// TwinCAT 3 PLC project Main
// ProgramVersion: 3.1.4023.0
// libraries:
//   Tc2_Standard, * (Beckhoff Automation GmbH)
//   Tc2_System, * (Beckhoff Automation GmbH)
//   Tc3_Module, * (Beckhoff Automation GmbH)
// project tree:
//   / PlcTask.TcTTO
//   POUs/ FB_Conveyor_SFC.TcPOU, FB_Conveyor_ST.TcPOU, FB_Coordinador_SFC.TcPOU, FB_Coordinador_ST.TcPOU, FB_Discharger_SFC.TcPOU, FB_Discharger_ST.TcPOU, FB_Elevator_SFC.TcPOU, FB_Elevator_ST.TcPOU, FB_Object_Template_ST.TcPOU, FB_Object_Template_SFC.TcPOU, MAIN.TcPOU
// real-time tasks:
//   TASK PlcTask: cycle T#10ms, priority 20, ADS port 350

CONFIGURATION Main
    RESOURCE PLC ON TwinCAT3
        TASK PlcTask(INTERVAL := T#10ms, PRIORITY := 20);
        PROGRAM MAIN WITH PlcTask : MAIN;
    END_RESOURCE
END_CONFIGURATION

// ---- POUs/MAIN.TcPOU
PROGRAM MAIN
VAR
	
Coordinador : FB_Coordinador_ST;

END_VAR

Coordinador();

END_PROGRAM

// ---- POUs/FB_Coordinador_ST.TcPOU
FUNCTION_BLOCK FB_Coordinador_ST EXTENDS FB_Object_Template_ST
VAR_INPUT
	//Discharger
	Tray_1 : BOOL; 
	Tray_2 : BOOL;
	
END_VAR
VAR_OUTPUT
	Fail : BOOL;
	B1   : BOOL;
	
END_VAR
VAR
	
	Discharger : FB_Discharger_ST;
	Elevators  : FB_Elevator_ST;
	Conveyors  : FB_Conveyor_ST;
	Production: FB_Coordinador_SFC;
	
END_VAR

IC := Discharger.IC AND Elevators.IC AND Conveyors.IC;
B1 := Selector(Tray_1,Tray_2);

Discharger(Execute:=Production.Discharger_Execute,
			Ack:=Production.Discharger_Ack,
			Reset:=Reset,
			Pause:=Pause,
			Tray_1:=Tray_1,
			Tray_2:=Tray_2
			);
			
Elevators.Elevator_B1 (Execute:=Production.Elevator_B1_Execute,
					  Ack:=Production.Elevator_B1_Ack,
					  SFCReset:=Reset,
					  SFCPause:=Pause,
					  );
					
Elevators.Elevator_B2 (Execute:=Production.Elevator_B2_Execute,
					  Ack:=Production.Elevator_B2_Ack,
					  SFCReset:=Reset,
					  SFCPause:=Pause,
					  );
					  
Elevators.Elevator_S (Execute:=Production.Elevator_S_Execute,
					  Ack:=Production.Elevator_S_Ack,
					  SFCReset:=Reset,
					  SFCPause:=Pause,
					  );
					  
Conveyors.Conveyors_B1  (Execute := Production.Conveyor_B1_Execute,
						Ack := Production.Conveyor_B1_Ack,
						SFCReset := Reset,
						SFCPause := Pause,
						);
						
Conveyors.Conveyors_B2  (Execute := Production.Conveyor_B2_Execute,
						Ack := Production.Conveyor_B2_Ack,
						SFCReset := Reset,
						SFCPause := Pause,
						);

Conveyors.Conveyor_S  (Execute := Production.Conveyor_S_Execute,
						Ack := Production.Conveyor_S_Ack,
						SFCReset := Reset,
						SFCPause := Pause,
						);

METHOD Selector : BOOL
VAR_INPUT
	
	Tray_1 : BOOL;
	Tray_2 : BOOL;

END_VAR
IF Tray_1 THEN
	Selector := TRUE;
ELSIF Tray_2 THEN
	Selector := FALSE;
END_IF
END_METHOD

END_FUNCTION_BLOCK

// ---- POUs/FB_Object_Template_ST.TcPOU
FUNCTION_BLOCK FB_Object_Template_ST
VAR_INPUT
	// Control variables
	Execute: BOOL;
	Ack: BOOL;
	Reset: BOOL; 
	Pause: BOOL;
	// Physical variables
	
END_VAR
VAR_OUTPUT
	//Control variables
	Ready: BOOL;
	Done: BOOL;
	//Physical Variables
	
END_VAR
VAR
	// Initial conditions
	IC: BOOL := TRUE;
END_VAR

END_FUNCTION_BLOCK

// ---- POUs/FB_Discharger_ST.TcPOU
FUNCTION_BLOCK FB_Discharger_ST EXTENDS FB_Object_Template_ST
VAR_INPUT
	Tray_1: BOOL; 
	Tray_2: BOOL;
	dcha_1 AT %I*: BOOL;
	dcha_2 AT %I*: BOOL;
	izda_1 AT %I*: BOOL;
	izda_2 AT %I*: BOOL;
	arriba AT %I*: BOOL;
	abajo  AT %I*: BOOL;
	cogido AT %I*: BOOL;
END_VAR
VAR_OUTPUT
	avanza_1 AT %Q*: BOOL;
	avanza_2 AT %Q*: BOOL;
	baja	 AT %Q*: BOOL;
	coge 	 AT %Q*: BOOL;
	Fail : BOOL;
	Timer : TON;
END_VAR
VAR
	Discharger : FB_Discharger_SFC;
END_VAR

//Define initial conditions
IC := izda_1 AND izda_2 AND arriba AND NOT cogido;
//Declare module
Discharger(Execute:=Execute,
		   Ack:=Ack,
		   SFCReset:=Reset,
		   SFCPause:=Pause,
		   IC:=IC,
		   Tray_1:=Tray_1,
		   Tray_2:=Tray_2,
		   dcha_1:=dcha_1,
		   dcha_2:=dcha_2,
		   izda_1:=izda_1,
		   izda_2:=izda_2,
		   arriba:=arriba,
		   abajo:=abajo,
		   cogido:=cogido,
);
		   
//Declare module actuators
Ready := Discharger.Ready;
Done := Discharger.Done;
avanza_1 := Discharger.avanza_1;
avanza_2 := Discharger.avanza_2;
baja := Discharger.baja;
coge := Discharger.coge;

END_FUNCTION_BLOCK

// ---- POUs/FB_Discharger_SFC.TcPOU
FUNCTION_BLOCK FB_Discharger_SFC EXTENDS FB_Object_Template_SFC
VAR_INPUT
	Tray_1: BOOL;
	Tray_2: BOOL;
	dcha_1: BOOL;
	dcha_2: BOOL;
	izda_1: BOOL;
	izda_2: BOOL;
	arriba: BOOL;
	abajo: BOOL;
	cogido: BOOL;
	Restore: BOOL;
END_VAR
VAR_OUTPUT
	avanza_1: BOOL;
	avanza_2: BOOL;
	baja: BOOL;
	coge: BOOL;
END_VAR
VAR
END_VAR

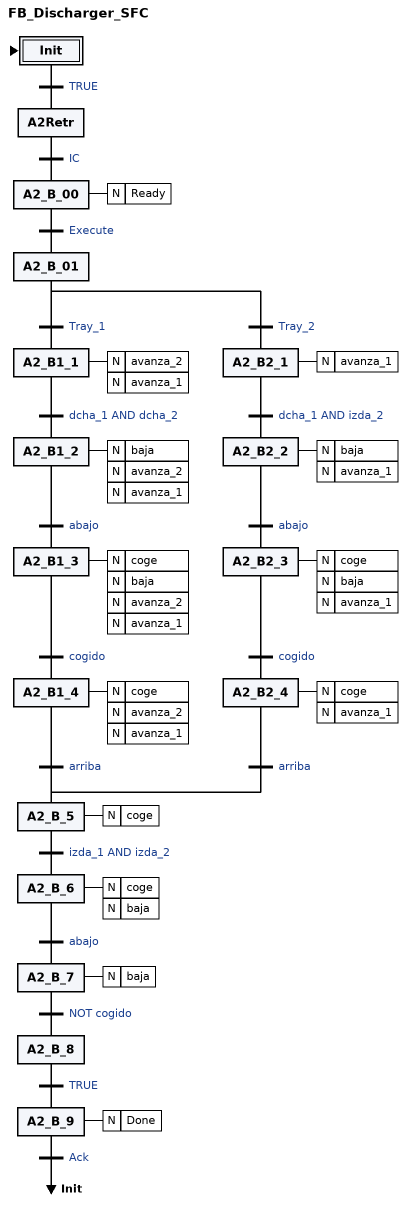
INITIAL_STEP Init:
END_STEP
TRANSITION FROM Init TO A2Retr
    := TRUE;
END_TRANSITION
STEP A2Retr:
END_STEP
TRANSITION FROM A2Retr TO A2_B_00
    := IC;
END_TRANSITION
STEP A2_B_00:
    Ready(N);
END_STEP
TRANSITION FROM A2_B_00 TO A2_B_01
    := Execute;
END_TRANSITION
STEP A2_B_01:
END_STEP
TRANSITION FROM A2_B_01 TO A2_B1_1
    := Tray_1;
END_TRANSITION
STEP A2_B1_1:
    avanza_2(N);
    avanza_1(N);
END_STEP
TRANSITION FROM A2_B1_1 TO A2_B1_2
    := dcha_1 AND dcha_2;
END_TRANSITION
STEP A2_B1_2:
    baja(N);
    avanza_2(N);
    avanza_1(N);
END_STEP
TRANSITION FROM A2_B1_2 TO A2_B1_3
    := abajo;
END_TRANSITION
STEP A2_B1_3:
    coge(N);
    baja(N);
    avanza_2(N);
    avanza_1(N);
END_STEP
TRANSITION FROM A2_B1_3 TO A2_B1_4
    := cogido;
END_TRANSITION
STEP A2_B1_4:
    coge(N);
    avanza_2(N);
    avanza_1(N);
END_STEP
TRANSITION FROM A2_B1_4 TO A2_B_5
    := arriba;
END_TRANSITION
TRANSITION FROM A2_B_01 TO A2_B2_1
    := Tray_2;
END_TRANSITION
STEP A2_B2_1:
    avanza_1(N);
END_STEP
TRANSITION FROM A2_B2_1 TO A2_B2_2
    := dcha_1 AND izda_2;
END_TRANSITION
STEP A2_B2_2:
    baja(N);
    avanza_1(N);
END_STEP
TRANSITION FROM A2_B2_2 TO A2_B2_3
    := abajo;
END_TRANSITION
STEP A2_B2_3:
    coge(N);
    baja(N);
    avanza_1(N);
END_STEP
TRANSITION FROM A2_B2_3 TO A2_B2_4
    := cogido;
END_TRANSITION
STEP A2_B2_4:
    coge(N);
    avanza_1(N);
END_STEP
TRANSITION FROM A2_B2_4 TO A2_B_5
    := arriba;
END_TRANSITION
STEP A2_B_5:
    coge(N);
END_STEP
TRANSITION FROM A2_B_5 TO A2_B_6
    := izda_1 AND izda_2;
END_TRANSITION
STEP A2_B_6:
    coge(N);
    baja(N);
END_STEP
TRANSITION FROM A2_B_6 TO A2_B_7
    := abajo;
END_TRANSITION
STEP A2_B_7:
    baja(N);
END_STEP
TRANSITION FROM A2_B_7 TO A2_B_8
    := NOT cogido;
END_TRANSITION
STEP A2_B_8:
END_STEP
TRANSITION FROM A2_B_8 TO A2_B_9
    := TRUE;
END_TRANSITION
STEP A2_B_9:
    Done(N);
END_STEP
TRANSITION FROM A2_B_9 TO Init
    := Ack;
END_TRANSITION

END_FUNCTION_BLOCK

// ---- POUs/FB_Object_Template_SFC.TcPOU
FUNCTION_BLOCK FB_Object_Template_SFC
VAR_INPUT
	// Control variables
	Execute: BOOL;
	Ack: BOOL;
	SFCReset: BOOL; 
	SFCPause: BOOL;
	IC: BOOL;
	// Physical variables
END_VAR
VAR_OUTPUT
	//Control variables
	Ready: BOOL;
	Done: BOOL;
	//Physical Variables
END_VAR
VAR
END_VAR

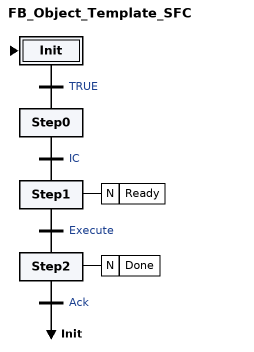
INITIAL_STEP Init:
END_STEP
TRANSITION FROM Init TO Step0
    := TRUE;
END_TRANSITION
STEP Step0:
END_STEP
TRANSITION FROM Step0 TO Step1
    := IC;
END_TRANSITION
STEP Step1:
    Ready(N);
END_STEP
TRANSITION FROM Step1 TO Step2
    := Execute;
END_TRANSITION
STEP Step2:
    Done(N);
END_STEP
TRANSITION FROM Step2 TO Init
    := Ack;
END_TRANSITION

END_FUNCTION_BLOCK

// ---- POUs/FB_Elevator_ST.TcPOU
FUNCTION_BLOCK FB_Elevator_ST EXTENDS FB_Object_Template_ST
VAR_INPUT
	
//Finales de Carrera
	END_Up_B1 AT %I*: BOOL;
	END_Down_B1 AT %I*: BOOL;
	END_Up_B2 AT %I*: BOOL;
	END_Down_B2 AT %I*: BOOL;
	END_Up_S AT %I*: BOOL;
	END_Down_S AT %I*: BOOL;
	END_Step AT %I*: BOOL;
	
//Señales de control
	Up_B1:BOOL;
	Down_B1:BOOL;
	Up_B2:BOOL;
	Down_B2:BOOL;
	Up_S:BOOL;
	Down_S:BOOL;
	Step:BOOL;

END_VAR
VAR_OUTPUT
	
//Acciones
	MOV_Up_B1 AT %Q*: BOOL;
	MOV_Down_B1 AT %Q*: BOOL;
	MOV_Up_B2 AT %Q*: BOOL;
	MOV_Down_B2 AT %Q*: BOOL;
	MOV_Up_S AT %Q*: BOOL;
	MOV_Down_S AT %Q*: BOOL;

END_VAR
VAR
	
	Elevator_B1: FB_Elevator_SFC;
	Elevator_B2: FB_Elevator_SFC;
	Elevator_S: FB_Elevator_SFC;

END_VAR

//Condicones Iniciales
IC := END_Down_B1 AND END_Down_B2 AND END_Up_S;

Elevator_B1(Execute:=Execute,
		   Ack:=Ack,
		   SFCReset:=Reset,
		   SFCPause:=Pause,
		   IC:=IC,
		   END_Up:=END_Up_B1,
		   END_Down:=END_Down_B1,
		   END_Step:=TRUE,
		   Up:=Up_B1,
		   Down:=Down_B1,
		   Step:=FALSE,	

);

Elevator_B2(Execute:=Execute,
		   Ack:=Ack,
		   SFCReset:=Reset,
		   SFCPause:=Pause,
		   IC:=IC,
		   END_Up:=END_Up_B2,
		   END_Down:=END_Down_B2,
		   END_Step:=TRUE,
		   Up:=Up_B2,
		   Down:=Down_B2,
		   Step:=FALSE,		   		

);

Elevator_S(Execute:=Execute,
		   Ack:=Ack,
		   SFCReset:=Reset,
		   SFCPause:=Pause,
		   IC:=IC,
		   END_Up:=END_Up_S,
		   END_Down:=END_Down_S,
		   END_Step:=END_Step,
		   Up:=Up_S,
		   Down:=Down_S,
		   Step:=Step,		   		

);
//Asignacion de acciones
	MOV_Up_B1:=Elevator_B1.MOV_Up;
	MOV_Down_B1:=Elevator_B1.MOV_Down;
	MOV_Up_B2:=Elevator_B2.MOV_Up;
	MOV_Down_B2:=Elevator_B2.MOV_Down;
	MOV_Up_S:=Elevator_S.MOV_Up;
	MOV_Down_S:=Elevator_S.MOV_Down OR Elevator_S.MOV_Step;

END_FUNCTION_BLOCK

// ---- POUs/FB_Elevator_SFC.TcPOU
FUNCTION_BLOCK FB_Elevator_SFC EXTENDS FB_Object_Template_SFC
VAR_INPUT

//Señales de accion
	Up:BOOL;
	Down:BOOL;
	Step:BOOL;
	
//Finales de carrera
	END_Up:BOOL;
	END_Down:BOOL;
	END_Step:BOOL;

END_VAR
VAR_OUTPUT
	
//Acciones
	MOV_Up:BOOL;
	MOV_Down:BOOL;
	MOV_Step:BOOL;

END_VAR
VAR
	
	T :TIME := T#0.5S;

END_VAR

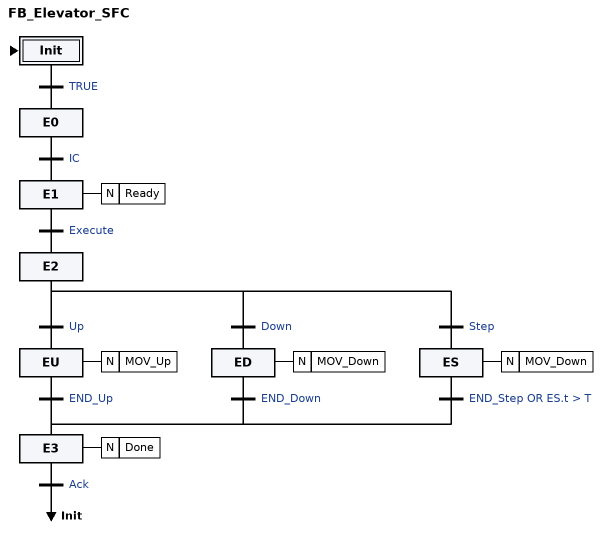
INITIAL_STEP Init:
END_STEP
TRANSITION FROM Init TO E0
    := TRUE;
END_TRANSITION
STEP E0:
END_STEP
TRANSITION FROM E0 TO E1
    := IC;
END_TRANSITION
STEP E1:
    Ready(N);
END_STEP
TRANSITION FROM E1 TO E2
    := Execute;
END_TRANSITION
STEP E2:
END_STEP
TRANSITION FROM E2 TO EU
    := Up;
END_TRANSITION
STEP EU:
    MOV_Up(N);
END_STEP
TRANSITION FROM EU TO E3
    := END_Up;
END_TRANSITION
TRANSITION FROM E2 TO ED
    := Down;
END_TRANSITION
STEP ED:
    MOV_Down(N);
END_STEP
TRANSITION FROM ED TO E3
    := END_Down;
END_TRANSITION
TRANSITION FROM E2 TO ES
    := Step;
END_TRANSITION
STEP ES:
    MOV_Down(N);
END_STEP
TRANSITION FROM ES TO E3
    := END_Step OR ES.t > T;
END_TRANSITION
STEP E3:
    Done(N);
END_STEP
TRANSITION FROM E3 TO Init
    := Ack;
END_TRANSITION

TRANSITION Execute:
Up OR Down OR Step;
END_TRANSITION

END_FUNCTION_BLOCK

// ---- POUs/FB_Conveyor_ST.TcPOU
FUNCTION_BLOCK FB_Conveyor_ST EXTENDS FB_Object_Template_ST
VAR_INPUT
	
// Finales de carrera
	END_Conv1_B1 AT %I* :BOOL;
	END_Conv2_B1 AT %I* :BOOL;
	END_Conv1_B2 AT %I* :BOOL;
	END_Conv2_B2 AT %I* :BOOL;
	END_Conv_S AT %I* :BOOL;

//Señales de control
	Produce_B1:BOOL;
	END_Produce_B1:BOOL;
	Produce_B2:BOOL;
	END_Produce_B2:BOOL;
	Take_Plate:BOOL;

END_VAR
VAR_OUTPUT
	
//Controles de las cintas
	MOV_Conv1_B1 AT %Q* :BOOL;
	MOV_Conv2_B1 AT %Q* :BOOL;
	MOV_Conv1_B2 AT %Q* :BOOL;
	MOV_Conv2_B2 AT %Q* :BOOL;
	MOV_Conv_S AT %Q* :BOOL;

END_VAR
VAR
	
	Conveyors_B1: FB_Conveyor_SFC;
	Conveyors_B2: FB_Conveyor_SFC;
	Conveyor_S: FB_Conveyor_SFC;


END_VAR

//Condiciones iniciales
IC := TRUE;
//Declaracion de las cintas
Conveyors_B1(Execute:=Execute,
		   Ack:=Ack,
		   SFCReset:=Reset,
		   SFCPause:=Pause,
		   IC:=IC,
		   END_Conv1 := END_Conv1_B1,
		   END_Conv2 := END_Conv2_B1,
		   Produce := Produce_B1,
		   END_Produce := END_Produce_B1
		   
);

Conveyors_B2(Execute:=Execute,
		   Ack:=Ack,
		   SFCReset:=Reset,
		   SFCPause:=Pause,
		   IC:=IC,
		   END_Conv1 := END_Conv1_B2,
		   END_Conv2 := END_Conv2_B2,
		   Produce := Produce_B2,
		   END_Produce := END_Produce_B2
		   
);

Conveyor_S(Execute:=Execute,
		   Ack:=Ack,
		   SFCReset:=Reset,
		   SFCPause:=Pause,
		   IC:=IC,
		   END_Conv1 := FALSE,
		   END_Conv2 := END_Conv_S,
		   Produce := FALSE,
		   END_Produce := Take_Plate
		   
);
		   
//Actuadores
	MOV_Conv1_B1 := Conveyors_B1.MOV_Conv1;
	MOV_Conv2_B1 := Conveyors_B1.MOV_Conv2;
	MOV_Conv1_B2 := Conveyors_B2.MOV_Conv1;
	MOV_Conv2_B2 := Conveyors_B2.MOV_Conv2;
	MOV_Conv_S := Conveyor_S.MOV_Conv2 OR Conveyor_S.MOV_Conv1;

END_FUNCTION_BLOCK

// ---- POUs/FB_Conveyor_SFC.TcPOU
FUNCTION_BLOCK FB_Conveyor_SFC EXTENDS FB_Object_Template_SFC
VAR_INPUT
	
	END_Conv2:BOOL;

END_VAR
VAR_OUTPUT
	
	MOV_Conv1:BOOL;
	MOV_Conv2:BOOL;

END_VAR
VAR
END_VAR

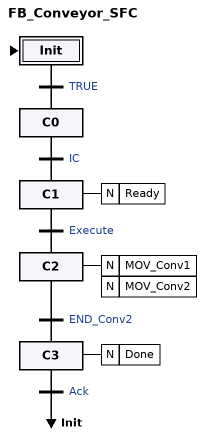
INITIAL_STEP Init:
END_STEP
TRANSITION FROM Init TO C0
    := TRUE;
END_TRANSITION
STEP C0:
END_STEP
TRANSITION FROM C0 TO C1
    := IC;
END_TRANSITION
STEP C1:
    Ready(N);
END_STEP
TRANSITION FROM C1 TO C2
    := Execute;
END_TRANSITION
STEP C2:
    MOV_Conv1(N);
    MOV_Conv2(N);
END_STEP
TRANSITION FROM C2 TO C3
    := END_Conv2;
END_TRANSITION
STEP C3:
    Done(N);
END_STEP
TRANSITION FROM C3 TO Init
    := Ack;
END_TRANSITION

END_FUNCTION_BLOCK

// ---- POUs/FB_Coordinador_SFC.TcPOU
FUNCTION_BLOCK FB_Coordinador_SFC EXTENDS FB_Object_Template_SFC;
VAR_INPUT
 
//Discharger
	Discharger_Ready: BOOL;
	Discharger_Done: BOOL;

	
//Elevador
	Elevator_B1_Ready:BOOL;
	Elevator_B2_Ready:BOOL;
	Elevator_S_Ready:BOOL;
	
	Elevator_B1_Done:BOOL;
	Elevator_B2_Done:BOOL;
	Elevator_S_Done:BOOL;

//Conveyors
	Conveyor_B1_Ready:BOOL;
	Conveyor_B2_Ready:BOOL;
	Conveyor_S_Ready:BOOL;
	
	Conveyor_B1_Done:BOOL;
	Conveyor_B2_Done:BOOL;
	Conveyor_S_Done:BOOL;
	
	Elevator_B1_END_Down:BOOL;
	Elevator_B2_END_Down:BOOL;
	Elevator_S_END_Down:BOOL;
	
	B1 :BOOL;

END_VAR
VAR_OUTPUT
	//Discharger
	Discharger_Ack: BOOL;
	Discharger_Execute: BOOL;
	
	//Elevador
	Elevator_B1_Execute:BOOL;
	Elevator_B2_Execute:BOOL;
	Elevator_S_Execute:BOOL;
	
	Elevator_B1_Up:BOOL;
	Elevator_B2_Up:BOOL;
	Elevator_S_Up:BOOL;
	
	Elevator_B1_Down:BOOL;
	Elevator_B2_Down:BOOL;
	Elevator_S_Down:BOOL;
	Elevator_S_Step:BOOL;
	
	Elevator_B1_Ack:BOOL;
	Elevator_B2_Ack:BOOL;
	Elevator_S_Ack:BOOL;

//Conveyor
	Conveyor_B1_Execute:BOOL;
	Conveyor_B2_Execute:BOOL;
	Conveyor_S_Execute:BOOL;
	
	Conveyor_B1_Ack:BOOL;
	Conveyor_B2_Ack:BOOL;
	Conveyor_S_Ack:BOOL;
	
	Conveyor_B1_Proces:BOOL;
	Conveyor_B2_Proces:BOOL;
	Conveyor_S_Dischar:BOOL;
	
END_VAR
VAR

//Cuenta de bandejas
	Count:INT;

END_VAR

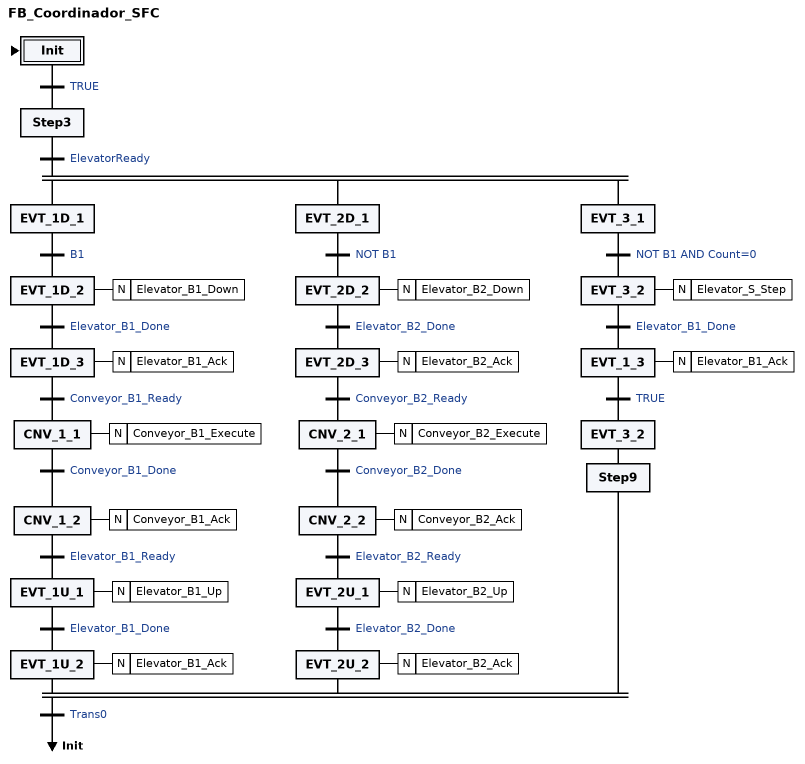
INITIAL_STEP Init:
END_STEP
TRANSITION FROM Init TO Step3
    := TRUE;
END_TRANSITION
STEP Step3:
END_STEP
TRANSITION FROM Step3 TO (EVT_1D_1, EVT_2D_1, EVT_3_1)
    := ElevatorReady;
END_TRANSITION
STEP EVT_1D_1:
END_STEP
TRANSITION FROM EVT_1D_1 TO EVT_1D_2
    := B1;
END_TRANSITION
STEP EVT_1D_2:
    Elevator_B1_Down(N);
END_STEP
TRANSITION FROM EVT_1D_2 TO EVT_1D_3
    := Elevator_B1_Done;
END_TRANSITION
STEP EVT_1D_3:
    Elevator_B1_Ack(N);
END_STEP
TRANSITION FROM EVT_1D_3 TO CNV_1_1
    := Conveyor_B1_Ready;
END_TRANSITION
STEP CNV_1_1:
    Conveyor_B1_Execute(N);
END_STEP
TRANSITION FROM CNV_1_1 TO CNV_1_2
    := Conveyor_B1_Done;
END_TRANSITION
STEP CNV_1_2:
    Conveyor_B1_Ack(N);
END_STEP
TRANSITION FROM CNV_1_2 TO EVT_1U_1
    := Elevator_B1_Ready;
END_TRANSITION
STEP EVT_1U_1:
    Elevator_B1_Up(N);
END_STEP
TRANSITION FROM EVT_1U_1 TO EVT_1U_2
    := Elevator_B1_Done;
END_TRANSITION
STEP EVT_1U_2:
    Elevator_B1_Ack(N);
END_STEP
STEP EVT_2D_1:
END_STEP
TRANSITION FROM EVT_2D_1 TO EVT_2D_2
    := NOT B1;
END_TRANSITION
STEP EVT_2D_2:
    Elevator_B2_Down(N);
END_STEP
TRANSITION FROM EVT_2D_2 TO EVT_2D_3
    := Elevator_B2_Done;
END_TRANSITION
STEP EVT_2D_3:
    Elevator_B2_Ack(N);
END_STEP
TRANSITION FROM EVT_2D_3 TO CNV_2_1
    := Conveyor_B2_Ready;
END_TRANSITION
STEP CNV_2_1:
    Conveyor_B2_Execute(N);
END_STEP
TRANSITION FROM CNV_2_1 TO CNV_2_2
    := Conveyor_B2_Done;
END_TRANSITION
STEP CNV_2_2:
    Conveyor_B2_Ack(N);
END_STEP
TRANSITION FROM CNV_2_2 TO EVT_2U_1
    := Elevator_B2_Ready;
END_TRANSITION
STEP EVT_2U_1:
    Elevator_B2_Up(N);
END_STEP
TRANSITION FROM EVT_2U_1 TO EVT_2U_2
    := Elevator_B2_Done;
END_TRANSITION
STEP EVT_2U_2:
    Elevator_B2_Ack(N);
END_STEP
STEP EVT_3_1:
END_STEP
TRANSITION FROM EVT_3_1 TO EVT_3_2
    := NOT B1 AND Count=0;
END_TRANSITION
STEP EVT_3_2:
    Elevator_S_Step(N);
END_STEP
TRANSITION FROM EVT_3_2 TO EVT_1_3
    := Elevator_B1_Done;
END_TRANSITION
STEP EVT_1_3:
    Elevator_B1_Ack(N);
END_STEP
TRANSITION FROM EVT_1_3 TO EVT_3_2
    := TRUE;
END_TRANSITION
STEP EVT_3_2:
END_STEP
// no transition between EVT_3_2 and Step9
STEP Step9:
END_STEP
TRANSITION FROM (EVT_1U_2, EVT_2U_2, Step9) TO Init
    := Trans0;
END_TRANSITION

TRANSITION ElevatorReady:
Elevator_B1_Ready OR Elevator_B2_Ready OR Elevator_S_Ready;
END_TRANSITION

END_FUNCTION_BLOCK
